// TIA Portal V19 export
ORGANIZATION_BLOCK "Main"   // OB2001, LAD, ProgramCycle
TITLE = "Main Program Sweep (Cycle)"
// This block calls the FB CallUnit which includes all further functionality of the unit.
// It reads the general global status and the safety status from the respective safety zone.
// It writes the unit status back to the DB Global.Data and the acknowledge information to the respetive safety zone.
// OB Main is a program cycle OB and is called depending on its number. For details, refer to the Automation Framework documentation.
// stored: AutoNumber false, IsIECCheckEnabled true, Namespace Unit, SetENOAutomatically true
   VAR_INPUT
      Initial_Call : Bool;   // Initial call of this OB
      Remanence : Bool;   // =True, if remanent data are available
   END_VAR
BEGIN

REGION Network 1: Call Unit
   // Call FB CallUnit and handover information from Global and Safety.
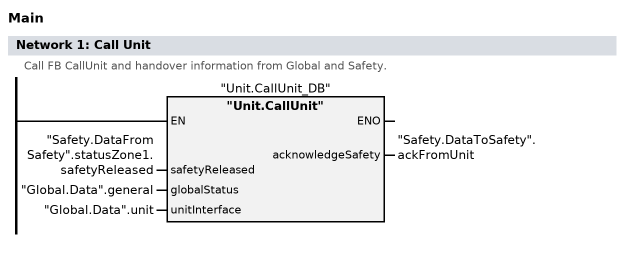
   RUNG wire#powerrail
      "Unit.CallUnit_DB"(safetyReleased := "Safety.DataFromSafety".statusZone1.safetyReleased, globalStatus := "Global.Data".general, unitInterface := "Global.Data".unit, acknowledgeSafety => "Safety.DataToSafety".ackFromUnit)
   END_RUNG
   // the same network as SCL:
   "Unit.CallUnit_DB"(safetyReleased := "Safety.DataFromSafety".statusZone1.safetyReleased,   // "Unit.CallUnit"
                      globalStatus := "Global.Data".general,
                      unitInterface := "Global.Data".unit,
                      acknowledgeSafety => "Safety.DataToSafety".ackFromUnit);
END_REGION
END_ORGANIZATION_BLOCK
